// Block: MwFakCalc_PS

DATA_BLOCK MwFakCalc_PS
{ S7_Optimized_Access := 'TRUE' }
VERSION : 0.1
   NON_RETAIN
   VAR
      StartMeasure : Bool;
      AuxStartMeasure : Bool;
      MeasureID : UInt;
      MeasuredValueG : LReal;
      MeasuredValueW : LReal;
   END_VAR

BEGIN
   // No initialization required
END_DATA_BLOCK
